PROGRAM MAIN
VAR

END_VAR

P_SingleADSRead();

END_PROGRAM

(* stored: Version 1.1.0.1, ProductVersion 3.1.4024.12
   POU MAIN: Id {0a750177-0d2a-4b56-b1a2-cbaaf547c1e4}, SpecialFunc None *)
